{attribute 'linkalways'} 
{attribute 'no_explicit_call' := 'This FB is a CLASS and must be accessed using methods or properties'}
{attribute 'enable_dynamic_creation'}
FUNCTION_BLOCK _SINT EXTENDS DatatypeBase
VAR
	localData : SINT;
	activeData : REFERENCE TO SINT REF= localData;
END_VAR

PROPERTY PUBLIC Address : PVOID
GET
Address := ADR(activeData);
END_GET
END_PROPERTY

METHOD PUBLIC ClearReference
VAR_INPUT
END_VAR
activeData REF= localData;
END_METHOD

METHOD PUBLIC Clone : I_Datatype
VAR
    pClone : POINTER TO _SINT;
END_VAR
pClone := __NEW(_SINT(InitialValue := Value));
Clone := pClone^;
END_METHOD

METHOD FB_init : BOOL
VAR_INPUT
	bInitRetains : BOOL; // if TRUE, the retain variables are initialized (warm start / cold start)
	bInCopyCode : BOOL;  // if TRUE, the instance afterwards gets moved into the copy code (online change)
	InitialValue : SINT;
END_VAR
localData := InitialValue;
END_METHOD

PROPERTY PUBLIC IecType : T_MAXSTRING
GET
IecType := 'SINT';
END_GET
END_PROPERTY

METHOD PUBLIC MakeReferenceTo
VAR_INPUT
	ReferenceTarget : REFERENCE TO SINT;
END_VAR
activeData REF= ReferenceTarget;
END_METHOD

METHOD PUBLIC SerializeWith
VAR_INPUT
	Serializer : I_Serializer;
END_VAR
Serializer.AddSint(activeData);
END_METHOD

PROPERTY PUBLIC Size : UDINT
GET
Size := SIZEOF(activeData);
END_GET
END_PROPERTY

METHOD TryDeserializeFrom : BOOL
VAR_INPUT
	Deserializer : I_Deserializer;
END_VAR
TryDeserializeFrom := Deserializer.TryGetSint(activeData);
END_METHOD

METHOD TryMakeReferenceTo : BOOL
VAR_INPUT
	Target : I_Datatype;
END_VAR
VAR
	pTargetData : POINTER TO SINT;
END_VAR
IF NOT (Target.IecType = IecType) THEN
	RETURN;
END_IF

pTargetData := Target.Address;
activeData REF= pTargetData^;
TryMakeReferenceTo := TRUE;
END_METHOD

PROPERTY PUBLIC Value : SINT
GET
Value := activeData;
END_GET
SET
activeData := Value;
END_SET
END_PROPERTY

END_FUNCTION_BLOCK

(* stored: Version 1.1.0.1, ProductVersion 3.1.4024.12
   POU _SINT: Id {63e171fa-a00a-01e6-2be5-267abd900597}, SpecialFunc None
   Folder Constructor: Id {47f4d29a-43d0-03a1-13ca-dd14b1c7c51e}
   Property Address: Id {9791cbf7-b868-03b9-0602-fa438c0662a3}
   Get Get: Id {05afff34-3f78-0219-08c4-5cf606369559}
   Method ClearReference: Id {0ee0dec8-402b-0a50-0108-8a719a9cd455}
   Method Clone: Id {d54602a1-4ce0-0c2f-2229-e1e2c5065e9b}
   Method FB_init: Id {8daaa383-0a7c-032b-3b8f-ee6d35797b8f}
   Property IecType: Id {6ddec637-949e-097d-3088-31c4dc70688d}
   Get Get: Id {183f2f01-44d1-02f1-32c4-770cb310d890}
   Method MakeReferenceTo: Id {bb0a599c-cb5d-0fce-2dd9-ed273e1f6c8b}
   Method SerializeWith: Id {af9a3f16-389e-0de7-0c47-39a628af0227}
   Property Size: Id {ab932130-909c-0109-3e51-462e921ffaae}
   Get Get: Id {e5bf6a81-d67d-0700-1099-8eeb7958a696}
   Method TryDeserializeFrom: Id {0b9e13ad-35fa-0b81-2484-57009f387016}
   Method TryMakeReferenceTo: Id {34f707c1-d40d-0e30-2757-816c497c7bf5}
   Property Value: Id {e0c01759-d0cd-09db-2dbf-737a2185225e}
   Get Get: Id {a32c337f-2a8f-0e65-398a-0e8c09d0d429}
   Set Set: Id {043eacc4-d935-067a-33da-0cdaa8251f35} *)
